(* PLC project FIO, Blank Blank 1.0 *)
(* stored: creationDateTime 2016-05-18T21:14:07, modificationDateTime 2017-03-27T11:16:15 *)

PROGRAM Scene1
  VAR
    sensor AT %IX0.0 : BOOL := true;
    conv_belt AT %QX0.0 : BOOL := true;
  END_VAR

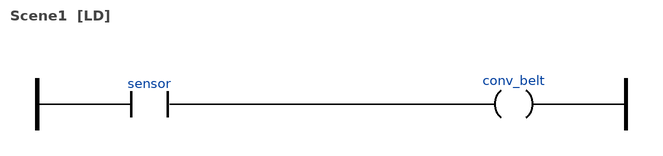
(* LD diagram, written out as Structured Text *)
conv_belt := sensor;
END_PROGRAM

CONFIGURATION Config
  RESOURCE Res ON PLC
    TASK TaskMain(INTERVAL := T#50ms, PRIORITY := 0);
    PROGRAM Inst WITH TaskMain : Scene1;
  END_RESOURCE
END_CONFIGURATION
